Omron CX-Programmer project NewProject (CX-Programmer 9.61)

# PLC Module_3_PIDAT: CP1H XA

## Global symbols (name address type ; comment)
202 CHANNEL  ; Float Level Sensor Input
210 CHANNEL  ; Servo Valve Output Control
D1 CHANNEL  ; Screen Display
D10 CHANNEL  ; GUI - C - SV
D100 CHANNEL  ; C - Set Point Value
D101 CHANNEL  ; C+1 - P Value
D102 CHANNEL  ; C+2 - I Value
D103 CHANNEL  ; C+3 - D Value
D104 CHANNEL  ; C+4 - Sampling Period
D105 CHANNEL  ; C+5 - PID Settings Designation
D106 CHANNEL  ; C+6 - MV Control
D107 CHANNEL  ; C+7 - MV Min. Value
D108 CHANNEL  ; C+8 - MV Max. Value
D109 CHANNEL  ; C+9 - Auto Tuning Settings
D11 CHANNEL  ; GUI - C+1 - P Value
D110 CHANNEL  ; C+10 - Limit-Cycle Hysteresis
D12 CHANNEL  ; GUI - C+2 - I Value
D13 CHANNEL  ; GUI - C+3 - D Value
D14 CHANNEL  ; GUI - C+4 - Sampling Period
D20 CHANNEL  ; Linear Function Offset
D21 CHANNEL  ; Delta Input Range
D22 CHANNEL  ; Delta Output Range
D23 CHANNEL  ; Max. Output
D24 CHANNEL  ; Min. Output
D27 CHANNEL  ; User Input Password
D28 CHANNEL  ; Correct Password
D30 CHANNEL  ; Min. Output
D31 CHANNEL  ; Min. Input
D32 CHANNEL  ; Max. Output
D33 CHANNEL  ; Max. Input
D35 CHANNEL  ; Min. Output
D36 CHANNEL  ; Min. Input
D37 CHANNEL  ; Max. Output
D38 CHANNEL  ; Max. Input
D40 CHANNEL  ; Tank Water Level BCD Equivalent
D41 CHANNEL  ; Set Point Level BCD Equivalent
D42 CHANNEL  ; Current Supplied to Servo Valve (mA)
D5 CHANNEL  ; User Input Password
D6 CHANNEL  ; Correct Password
T0000 BOOL  ; Initialization Delay
T0001 BOOL  ; Title Screen Delay
T0002 BOOL  ; Password Screen Shift Delay

## Program Tank_Water_Control_by_PIDAT (cyclic task 0)
Local symbols
AUTO_TUNING 15.00 BOOL  ; 15.00 - AUTO_TUNING
Controller 11.00 BOOL  ; 11.00 - Controller
D_Value_Control 18.00 BOOL  ; 18.00 - D_Value_Control
GUI_Start 5.00 BOOL  ; 5.00 - GUI_Start
GUI_Stop 6.00 BOOL  ; 6.00 - GUI_Stop
I_Value_Control 17.00 BOOL  ; 17.00 - I_Value_Control
PB_Start 0.00 BOOL  ; 0.00 - PB_Start
PB_Stop 1.00 BOOL  ; 1.00 - PB_Stop
PID_Button_Control 11.03 BOOL  ; 11.03 - PID_Button_Control
PID_Controller 14.00 BOOL  ; 14.00 - PID_Controller
PI_Button_Control 11.02 BOOL  ; 11.02 - PI_Button_Control
PI_Controller 13.00 BOOL  ; 13.00 - PI_Controller
P_Button_Control 11.01 BOOL  ; 11.01 - P_Button_Control
P_Controller 12.00 BOOL  ; 12.00 - P_Controller
P_Value_Control 16.00 BOOL  ; 16.00 - P_Value_Control
START 10.00 BOOL  ; 10.00 - START
Submit_Password 2.00 BOOL  ; 2.00 - Submit_Password

### Section Initialization_Section

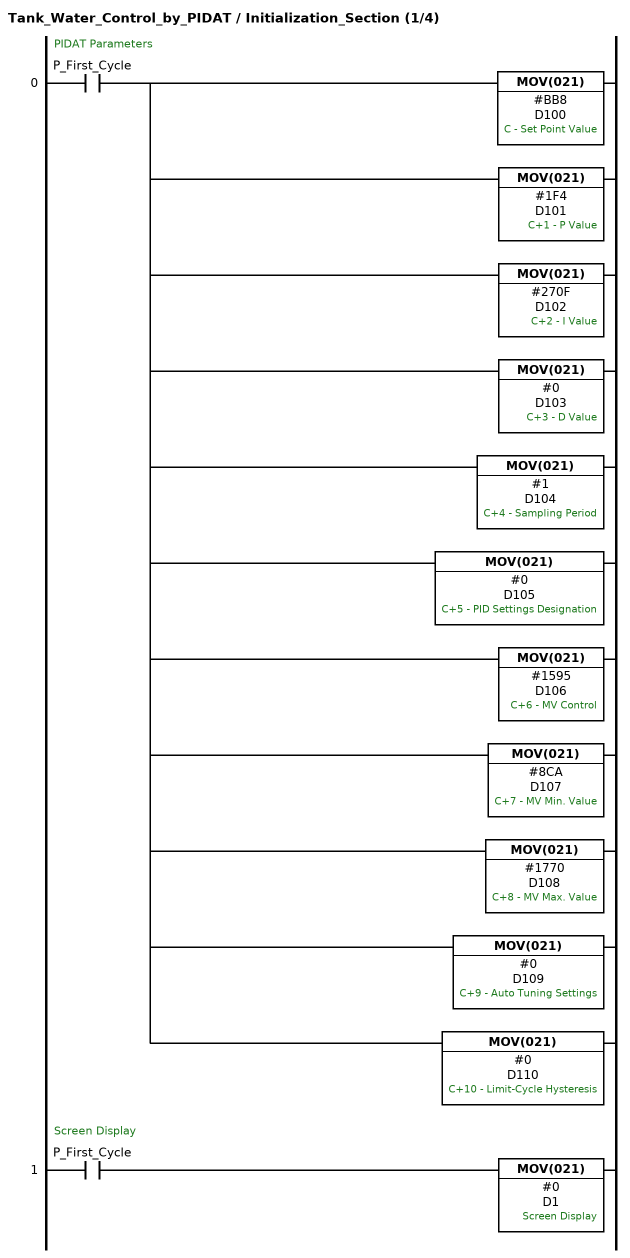
; rung 0: PIDAT Parameters
LD P_First_Cycle
MOV(021) #BB8 D100  ; C - Set Point Value
MOV(021) #1F4 D101  ; C+1 - P Value
MOV(021) #270F D102  ; C+2 - I Value
MOV(021) #0 D103  ; C+3 - D Value
MOV(021) #1 D104  ; C+4 - Sampling Period
MOV(021) #0 D105  ; C+5 - PID Settings Designation
MOV(021) #1595 D106  ; C+6 - MV Control
MOV(021) #8CA D107  ; C+7 - MV Min. Value
MOV(021) #1770 D108  ; C+8 - MV Max. Value
MOV(021) #0 D109  ; C+9 - Auto Tuning Settings
MOV(021) #0 D110  ; C+10 - Limit-Cycle Hysteresis
; rung 1: Screen Display
LD P_First_Cycle
MOV(021) #0 D1  ; Screen Display

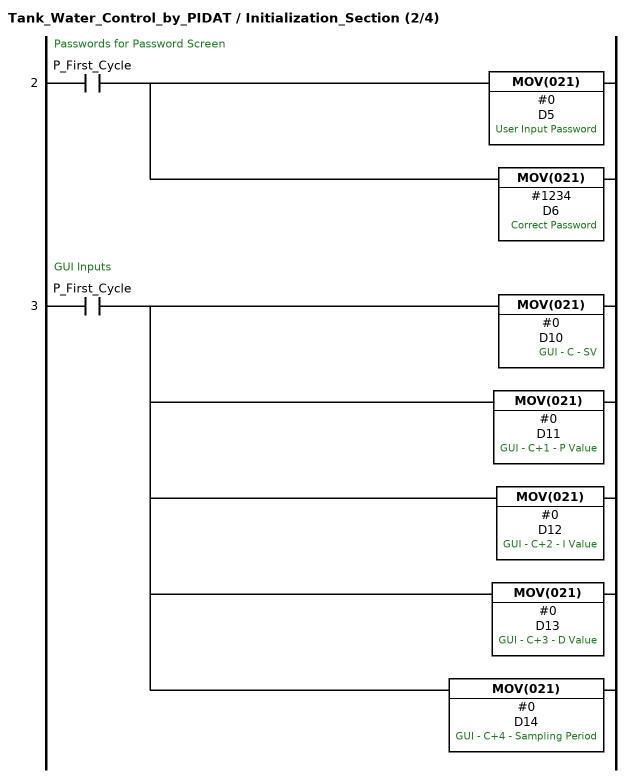
; rung 2: Passwords for Password Screen
LD P_First_Cycle
MOV(021) #0 D5  ; User Input Password
MOV(021) #1234 D6  ; Correct Password
; rung 3: GUI Inputs
LD P_First_Cycle
MOV(021) #0 D10  ; GUI - C - SV
MOV(021) #0 D11  ; GUI - C+1 - P Value
MOV(021) #0 D12  ; GUI - C+2 - I Value
MOV(021) #0 D13  ; GUI - C+3 - D Value
MOV(021) #0 D14  ; GUI - C+4 - Sampling Period

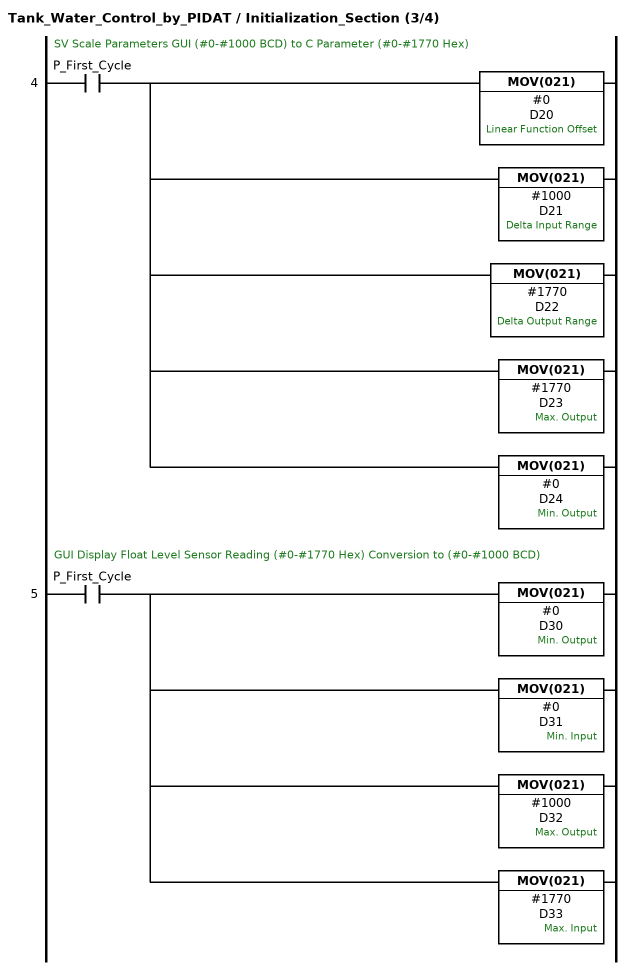
; rung 4: SV Scale Parameters GUI (#0-#1000 BCD) to C Parameter (#0-#1770 Hex)
LD P_First_Cycle
MOV(021) #0 D20  ; Linear Function Offset
MOV(021) #1000 D21  ; Delta Input Range
MOV(021) #1770 D22  ; Delta Output Range
MOV(021) #1770 D23  ; Max. Output
MOV(021) #0 D24  ; Min. Output
; rung 5: GUI Display Float Level Sensor Reading (#0-#1770 Hex) Conversion to (#0-#1000 BCD)
LD P_First_Cycle
MOV(021) #0 D30  ; Min. Output
MOV(021) #0 D31  ; Min. Input
MOV(021) #1000 D32  ; Max. Output
MOV(021) #1770 D33  ; Max. Input

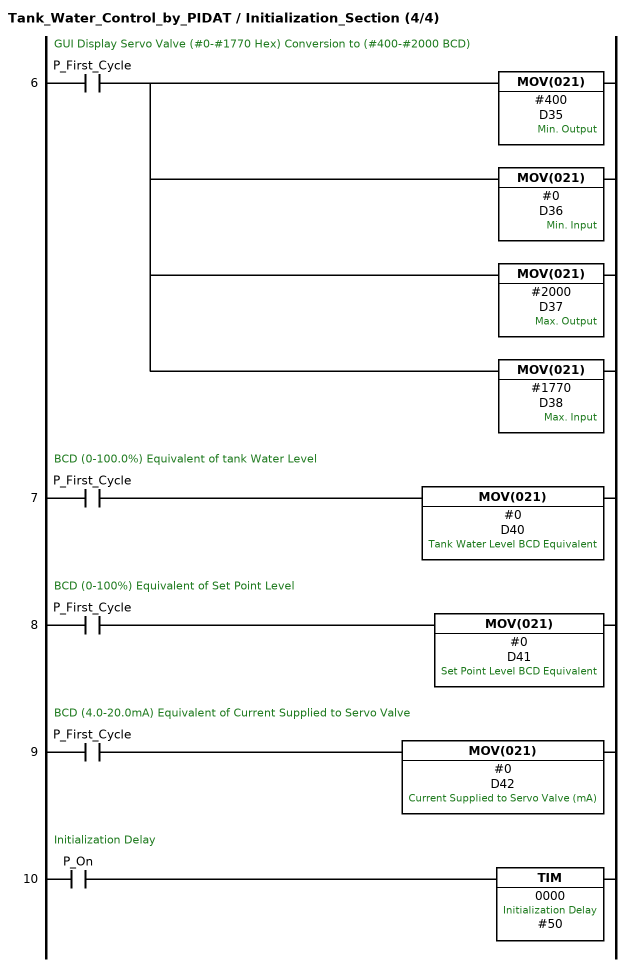
; rung 6: GUI Display Servo Valve (#0-#1770 Hex) Conversion to (#400-#2000 BCD)
LD P_First_Cycle
MOV(021) #400 D35  ; Min. Output
MOV(021) #0 D36  ; Min. Input
MOV(021) #2000 D37  ; Max. Output
MOV(021) #1770 D38  ; Max. Input
; rung 7: BCD (0-100.0%) Equivalent of tank Water Level
LD P_First_Cycle
MOV(021) #0 D40  ; Tank Water Level BCD Equivalent
; rung 8: BCD (0-100%) Equivalent of Set Point Level
LD P_First_Cycle
MOV(021) #0 D41  ; Set Point Level BCD Equivalent
; rung 9: BCD (4.0-20.0mA) Equivalent of Current Supplied to Servo Valve
LD P_First_Cycle
MOV(021) #0 D42  ; Current Supplied to Servo Valve (mA)
; rung 10: Initialization Delay
LD P_On
TIM 0000 #50  ; Initialization Delay

### Section Screen_Control_Section

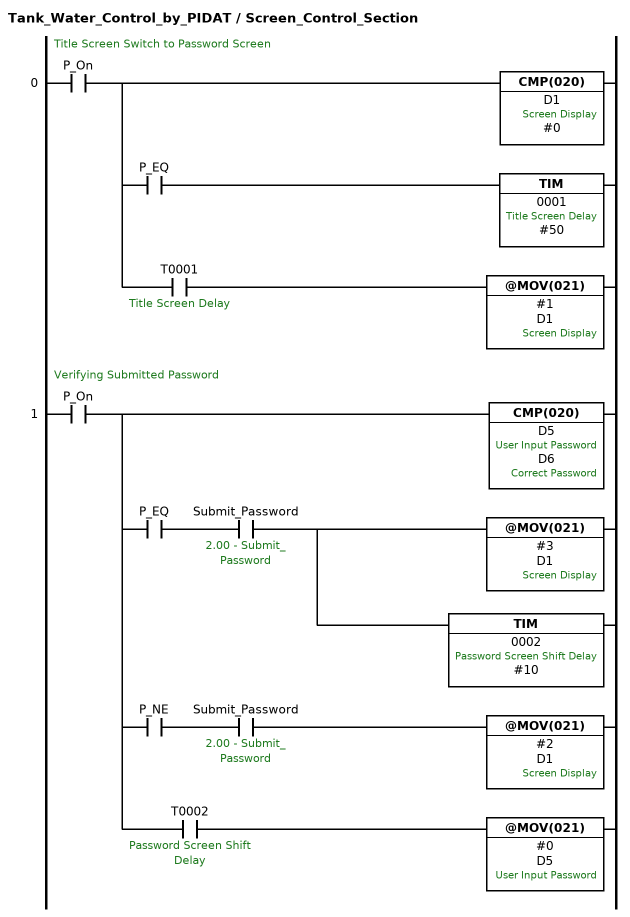
; rung 0: Title Screen Switch to Password Screen
LD P_On
OUT TR0
CMP(020) D1 #0  ; Screen Display
AND P_EQ
TIM 0001 #50  ; Title Screen Delay
LD TR0
AND T0001  ; Title Screen Delay
@MOV(021) #1 D1  ; Screen Display
; rung 1: Verifying Submitted Password
LD P_On
OUT TR0
CMP(020) D5 D6  ; User Input Password, Correct Password
AND P_EQ
AND Submit_Password  ; 2.00 - Submit_Password
@MOV(021) #3 D1  ; Screen Display
TIM 0002 #10  ; Password Screen Shift Delay
LD TR0
AND P_NE
AND Submit_Password  ; 2.00 - Submit_Password
@MOV(021) #2 D1  ; Screen Display
LD TR0
AND T0002  ; Password Screen Shift Delay
@MOV(021) #0 D5  ; User Input Password

### Section Main_Program_Section

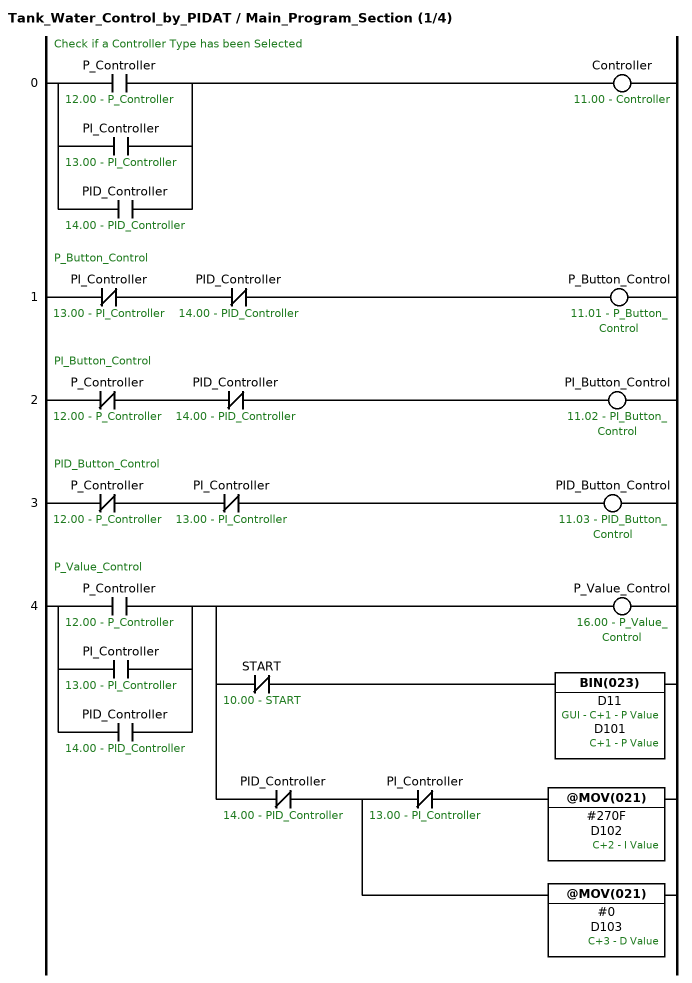
; rung 0: Check if a Controller Type has been Selected
LD P_Controller  ; 12.00 - P_Controller
OR PI_Controller  ; 13.00 - PI_Controller
OR PID_Controller  ; 14.00 - PID_Controller
OUT Controller  ; 11.00 - Controller
; rung 1: P_Button_Control
LDNOT PI_Controller  ; 13.00 - PI_Controller
ANDNOT PID_Controller  ; 14.00 - PID_Controller
OUT P_Button_Control  ; 11.01 - P_Button_Control
; rung 2: PI_Button_Control
LDNOT P_Controller  ; 12.00 - P_Controller
ANDNOT PID_Controller  ; 14.00 - PID_Controller
OUT PI_Button_Control  ; 11.02 - PI_Button_Control
; rung 3: PID_Button_Control
LDNOT P_Controller  ; 12.00 - P_Controller
ANDNOT PI_Controller  ; 13.00 - PI_Controller
OUT PID_Button_Control  ; 11.03 - PID_Button_Control
; rung 4: P_Value_Control
LD P_Controller  ; 12.00 - P_Controller
OR PI_Controller  ; 13.00 - PI_Controller
OR PID_Controller  ; 14.00 - PID_Controller
OUT TR0
OUT P_Value_Control  ; 16.00 - P_Value_Control
ANDNOT START  ; 10.00 - START
BIN(023) D11 D101  ; GUI - C+1 - P Value, C+1 - P Value
LD TR0
ANDNOT PID_Controller  ; 14.00 - PID_Controller
OUT TR0
ANDNOT PI_Controller  ; 13.00 - PI_Controller
@MOV(021) #270F D102  ; C+2 - I Value
LD TR0
@MOV(021) #0 D103  ; C+3 - D Value

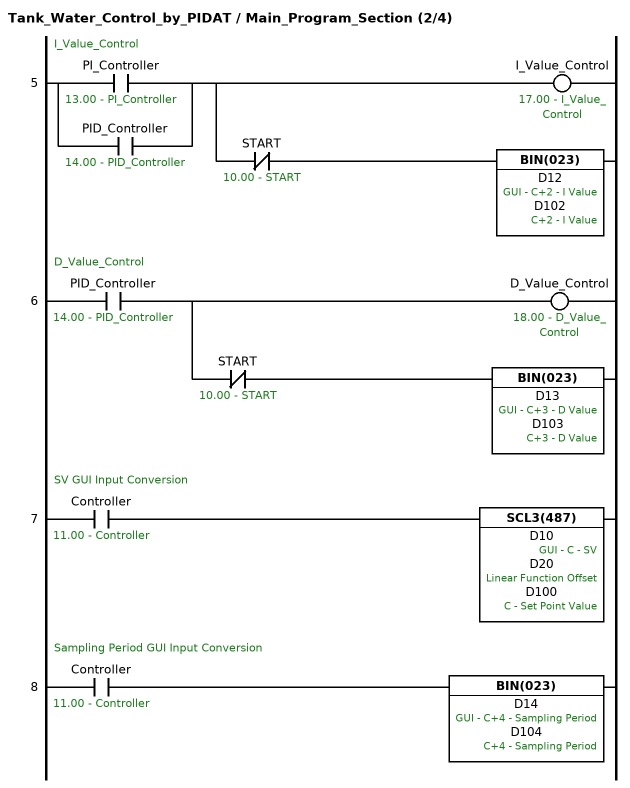
; rung 5: I_Value_Control
LD PI_Controller  ; 13.00 - PI_Controller
OR PID_Controller  ; 14.00 - PID_Controller
OUT I_Value_Control  ; 17.00 - I_Value_Control
ANDNOT START  ; 10.00 - START
BIN(023) D12 D102  ; GUI - C+2 - I Value, C+2 - I Value
; rung 6: D_Value_Control
LD PID_Controller  ; 14.00 - PID_Controller
OUT D_Value_Control  ; 18.00 - D_Value_Control
ANDNOT START  ; 10.00 - START
BIN(023) D13 D103  ; GUI - C+3 - D Value, C+3 - D Value
; rung 7: SV GUI Input Conversion
LD Controller  ; 11.00 - Controller
SCL3(487) D10 D20 D100  ; GUI - C - SV, Linear Function Offset, C - Set Point Value
; rung 8: Sampling Period GUI Input Conversion
LD Controller  ; 11.00 - Controller
BIN(023) D14 D104  ; GUI - C+4 - Sampling Period, C+4 - Sampling Period

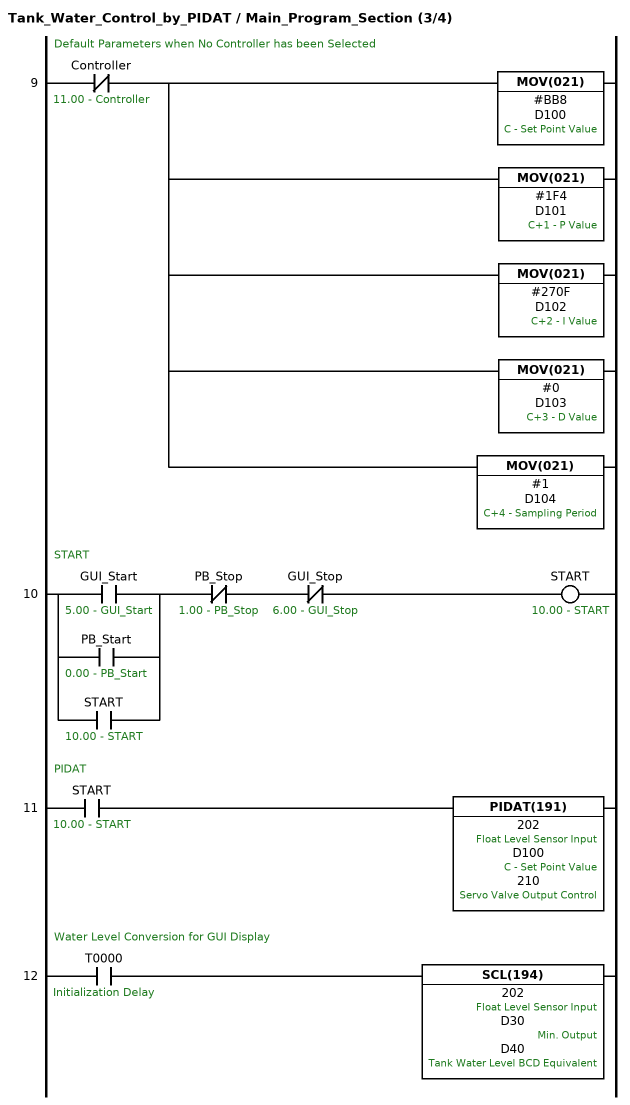
; rung 9: Default Parameters when No Controller has been Selected
LDNOT Controller  ; 11.00 - Controller
MOV(021) #BB8 D100  ; C - Set Point Value
MOV(021) #1F4 D101  ; C+1 - P Value
MOV(021) #270F D102  ; C+2 - I Value
MOV(021) #0 D103  ; C+3 - D Value
MOV(021) #1 D104  ; C+4 - Sampling Period
; rung 10: START
LD GUI_Start  ; 5.00 - GUI_Start
OR PB_Start  ; 0.00 - PB_Start
OR START  ; 10.00 - START
ANDNOT PB_Stop  ; 1.00 - PB_Stop
ANDNOT GUI_Stop  ; 6.00 - GUI_Stop
OUT START  ; 10.00 - START
; rung 11: PIDAT
LD START  ; 10.00 - START
PIDAT(191) 202 D100 210  ; Float Level Sensor Input, C - Set Point Value, Servo Valve Output Control
; rung 12: Water Level Conversion for GUI Display
LD T0000  ; Initialization Delay
SCL(194) 202 D30 D40  ; Float Level Sensor Input, Min. Output, Tank Water Level BCD Equivalent

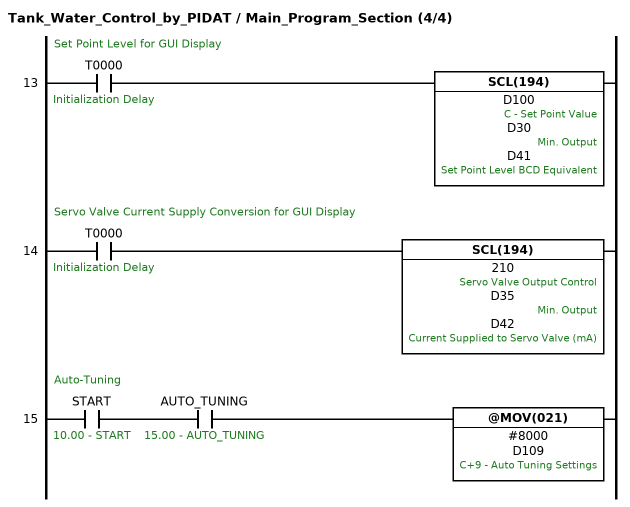
; rung 13: Set Point Level for GUI Display
LD T0000  ; Initialization Delay
SCL(194) D100 D30 D41  ; C - Set Point Value, Min. Output, Set Point Level BCD Equivalent
; rung 14: Servo Valve Current Supply Conversion for GUI Display
LD T0000  ; Initialization Delay
SCL(194) 210 D35 D42  ; Servo Valve Output Control, Min. Output, Current Supplied to Servo Valve (mA)
; rung 15: Auto-Tuning
LD START  ; 10.00 - START
AND AUTO_TUNING  ; 15.00 - AUTO_TUNING
@MOV(021) #8000 D109  ; C+9 - Auto Tuning Settings

### Section END
; rung 0
END(001)